TEXTLIST MachineState
  10 = 'Off'
  20 = 'Run'
  0 = 'Init'
   = ''
END_TEXTLIST

(* stored: Version 1.1.0.1, ProductVersion 3.1.4024.3
   TextList MachineState: Id {6e6451a3-d904-452f-bd36-f404b5e10305} *)
